{attribute addProperty BoxType "ELM3002-0000-0016"}
{attribute addProperty Id "StatusAT %I*Status_6A40DED4324"}
{attribute addProperty CRC "3480367792"}
{attribute addProperty SizeInBites "32"}
{attribute addProperty SizeInBytes "4"}
TYPE PAI_Status_Channel_CF7232B0 :
STRUCT
	{attribute addProperty Name "Status"}
	Status AT %I* : Status_6A40DED4;
END_STRUCT
END_TYPE

(* stored: Version 1.2.0.0, ProductVersion 3.1.4024.9
   DUT PAI_Status_Channel_CF7232B0: Id {66595926-13c6-47d9-b226-bae6bd46cf4d} *)
